(* CoDeSys 2.3.9.59 project: PD3.pro *)
(* Libraries: Standard.lib, SYSLIBCALLBACK.LIB *)

(* PLC configuration (modules and I/O channels)
Configuration EC4P-200 [Root] node -1, in %IB0 out %QB0 {EC4P_RestartPwrOn = WARMSTART; EC4P_MaxCycleTime = 20; EC4P_Com1BaudRate = 38400; EC4P_CAN1BaudRate = 125KBaud; EC4P_RoutingId = 127; EC4P_EasyNetId = 1; EC4P_EasyNetCfg = 0; EC4P_EasyNetCycleTime = 50; EC4P_RoutingChannel = CAN1; EC4P_IPFlags = 0; EC4P_IPAddress = 0; EC4P_SubNetMask = 0; EC4P_DefaultGateway = 0; EC4P_SummerWinterFlags = 0; EC4P_SummerWinterRule1 = 0; EC4P_SummerWinterRule2 = 0}
  Local I/O [EC4P_LocalIO] node 0, in %IB0 out %QB0 {EC4P_LocalInt = 0}
    I1 AT %IX0.0 [LocalBitInput] Input I1
    I2 AT %IX0.1 [LocalBitInput] Input I2
    I3 AT %IX0.2 [LocalBitInput] Input I3
    I4 AT %IX0.3 [LocalBitInput] Input I4
    I5 AT %IX0.4 [LocalBitInput] Input I5
    I6 AT %IX0.5 [LocalBitInput] Input I6
    I7 AT %IX0.6 [LocalBitInput] Input I7
    I8 AT %IX0.7 [LocalBitInput] Input I8
    I9 AT %IX1.0 [LocalBitInput] Input I9
    I10 AT %IX1.1 [LocalBitInput] Input I10
    I11 AT %IX1.2 [LocalBitInput] Input I11
    I12 AT %IX1.3 [LocalBitInput] Input I12
    I13 AT %IX1.4 [LocalDiagInput] Diagnostic Input I13
    I14 AT %IX1.5 [LocalDiagInput] Diagnostic Input I14
    I15 AT %IX1.6 [LocalDiagInput] Diagnostic Input I15
    I16 AT %IX1.7 [LocalDiagInput] Diagnostic Input I16
    I7_Analog AT %IW2 [LocalAnalogIn] Input I7, 10Bit, 0-10VDC
    I8_Analog AT %IW4 [LocalAnalogIn] Input I8, 10Bit, 0-10VDC
    I11_Analog AT %IW6 [LocalAnalogIn] Input I11, 10Bit, 0-10VDC
    I12_Analog AT %IW8 [LocalAnalogIn] Input I12, 10Bit, 0-10VDC
    Transistor Outputs [EC4P_TOutputs] node 0, in %IB10 out %QB0
      Q1 AT %QX0.0 [LocalBitOutput] Transistor-Output Q1
      Q2 AT %QX0.1 [LocalBitOutput] Transistor-Output Q2
      Q3 AT %QX0.2 [LocalBitOutput] Transistor-Output Q3
      Q4 AT %QX0.3 [LocalBitOutput] Transistor-Output Q4
      Q5 AT %QX0.4 [LocalBitOutput] Transistor-Output Q5
      Q6 AT %QX0.5 [LocalBitOutput] Transistor-Output Q6
      Q7 AT %QX0.6 [LocalBitOutput] Transistor-Output Q7
      Q8 AT %QX0.7 [LocalBitOutput] Transistor-Output Q8
    No Analog Output [EC4P_NoAnalogOutput] node 1, in %IB10 out %QB1
    No Keys [EC4P_NoKeys] node 2, in %IB10 out %QB1
    No Counter [EC4P_NoCounter] node 3, in %IB10 out %QB1
  Extension [EC4P_Extension] node 1, in %IB10 out %QB1
    No Extension [EC4P_NoExtension] node 0, in %IB10 out %QB1
*)

(* POU PLC_PRG, LD *)
PROGRAM PLC_PRG
VAR
	A: BOOL;
	B: BOOL;
	C: BOOL;
	D: BOOL;
	E: BOOL;
	ctu1: CTU;
	counter: INT;
	timer: BOOL;
	res: BOOL;
	TON1: TON;
	init: BOOL;
	tim: BOOL;
	TON2: TON;
	TON3: TON;
	temp: BOOL;
	t1: TIME;
	t2: TIME;
	TOF1: TOF;
	set_1: BOOL;
	set_2: BOOL;
	set_3: BOOL;
	set_4: BOOL;
	set_5: BOOL;
END_VAR
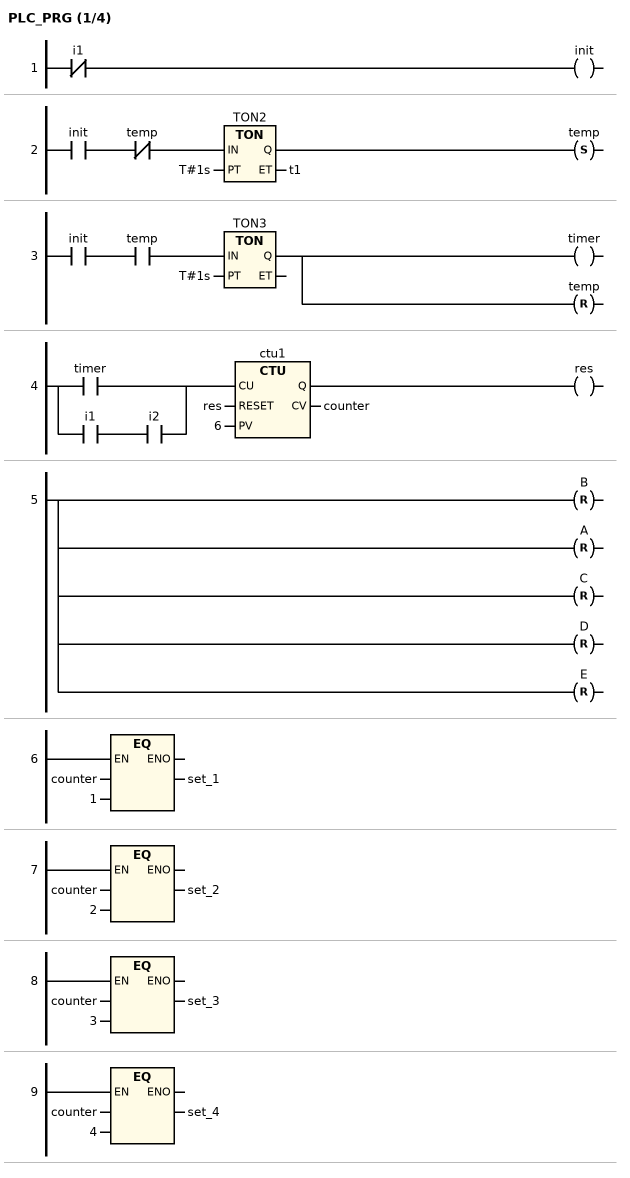
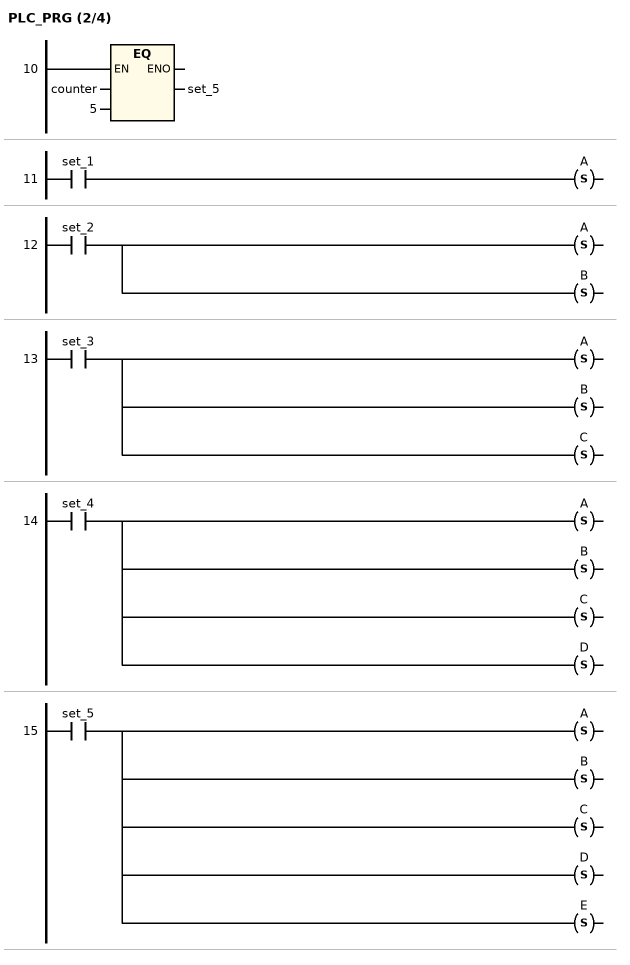
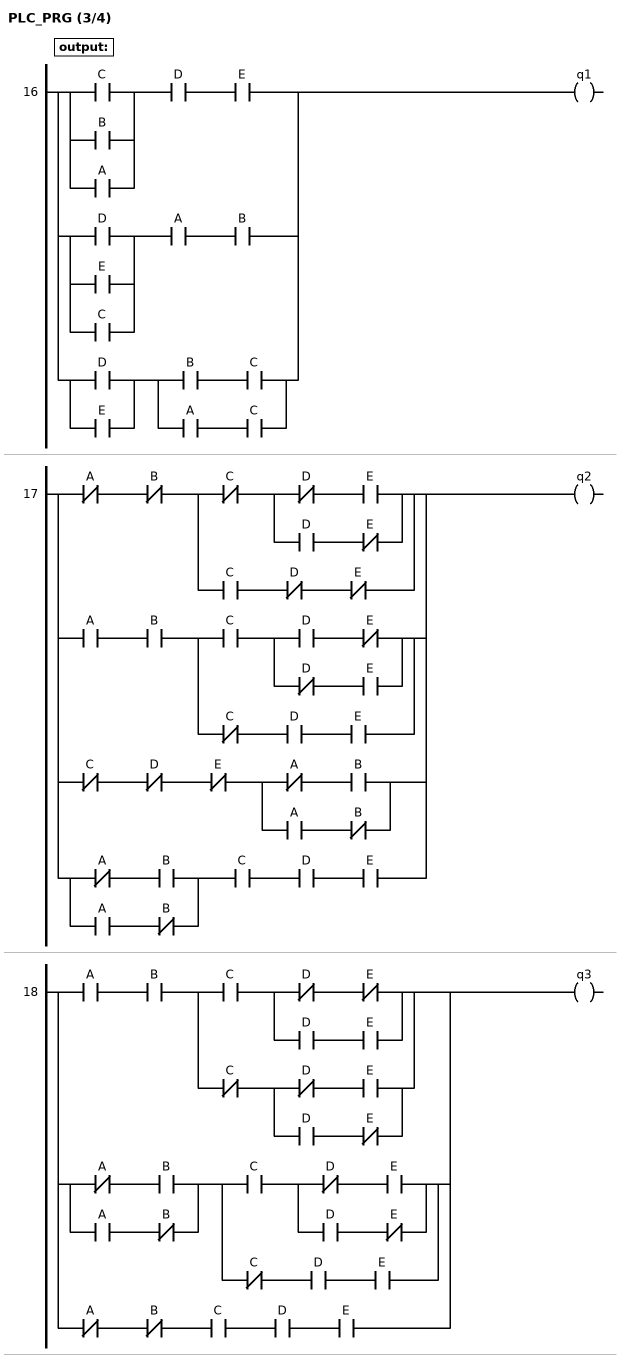
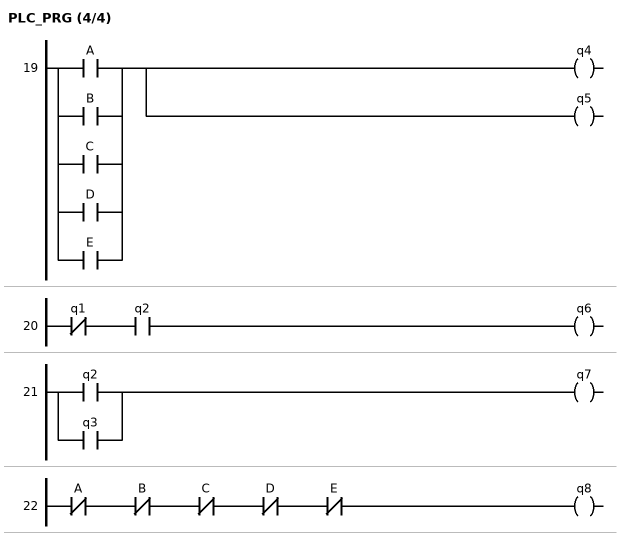
_LD_ (* Ladder Diagram *)
NETWORK 1
	[/i1] --- (init)
NETWORK 2
	[init] - [/temp] - TON2:TON(IN: *, PT: T#1s, ET => t1) --- (S temp)
NETWORK 3
	[init] - [temp] - TON3:TON(IN: *, PT: T#1s) --- (timer) (R temp)
NETWORK 4
	{ [timer] | [i1] - [i2] } - ctu1:CTU(CU: *, RESET: res, PV: 6, CV => counter) --- (res)
NETWORK 5
	* --- (R B) (R A) (R C) (R D) (R E)
NETWORK 6
	*
		EN --- EQ(counter, 1) => set_1
NETWORK 7
	*
		EN --- EQ(counter, 2) => set_2
NETWORK 8
	*
		EN --- EQ(counter, 3) => set_3
NETWORK 9
	*
		EN --- EQ(counter, 4) => set_4
NETWORK 10
	*
		EN --- EQ(counter, 5) => set_5
NETWORK 11
	[set_1] --- (S A)
NETWORK 12
	[set_2] --- (S A) (S B)
NETWORK 13
	[set_3] --- (S A) (S B) (S C)
NETWORK 14
	[set_4] --- (S A) (S B) (S C) (S D)
NETWORK 15
	[set_5] --- (S A) (S B) (S C) (S D) (S E)
NETWORK 16 output::
	{ { [C] | [B] | [A] } - [D] - [E] | { [D] | [E] | [C] } - [A] - [B] | { [D] | [E] } - { [B] - [C] | [A] - [C] } } --- (q1)
NETWORK 17
	{ [/A] - [/B] - { [/C] - { [/D] - [E] | [D] - [/E] } | [C] - [/D] - [/E] } | [A] - [B] - { [C] - { [D] - [/E] | [/D] - [E] } | [/C] - [D] - [E] } | [/C] - [/D] - [/E] - { [/A] - [B] | [A] - [/B] } | { [/A] - [B] | [A] - [/B] } - [C] - [D] - [E] } --- (q2)
NETWORK 18
	{ [A] - [B] - { [C] - { [/D] - [/E] | [D] - [E] } | [/C] - { [/D] - [E] | [D] - [/E] } } | { [/A] - [B] | [A] - [/B] } - { [C] - { [/D] - [E] | [D] - [/E] } | [/C] - [D] - [E] } | [/A] - [/B] - [C] - [D] - [E] } --- (q3)
NETWORK 19
	{ [A] | [B] | [C] | [D] | [E] } --- (q4) (q5)
NETWORK 20
	[/q1] - [q2] --- (q6)
NETWORK 21
	{ [q2] | [q3] } --- (q7)
NETWORK 22
	[/A] - [/B] - [/C] - [/D] - [/E] --- (q8)
_END_LD_
(* the same logic as Structured Text *)
(* Network 1 *)
init := NOT i1;
(* Network 2 *)
TON2(IN := init AND NOT temp, PT := T#1s);
t1 := TON2.ET;
IF TON2.Q THEN temp := TRUE; END_IF;
(* Network 3 *)
TON3(IN := init AND temp, PT := T#1s);
timer := TON3.Q;
IF TON3.Q THEN temp := FALSE; END_IF;
(* Network 4 *)
ctu1(CU := timer OR i1 AND i2, RESET := res, PV := 6);
counter := ctu1.CV;
res := ctu1.Q;
(* Network 5 *)
B := FALSE;
A := FALSE;
C := FALSE;
D := FALSE;
E := FALSE;
(* Network 6 *)
set_1 := counter = 1;
(* Network 7 *)
set_2 := counter = 2;
(* Network 8 *)
set_3 := counter = 3;
(* Network 9 *)
set_4 := counter = 4;
(* Network 10 *)
set_5 := counter = 5;
(* Network 11 *)
IF set_1 THEN A := TRUE; END_IF;
(* Network 12 *)
IF set_2 THEN A := TRUE; B := TRUE; END_IF;
(* Network 13 *)
IF set_3 THEN A := TRUE; B := TRUE; C := TRUE; END_IF;
(* Network 14 *)
IF set_4 THEN A := TRUE; B := TRUE; C := TRUE; D := TRUE; END_IF;
(* Network 15 *)
IF set_5 THEN A := TRUE; B := TRUE; C := TRUE; D := TRUE; E := TRUE; END_IF;
(* Network 16 *)
(* label: output: *)
q1 := (C OR B OR A) AND D AND E OR (D OR E OR C) AND A AND B OR (D OR E) AND (B AND C OR A AND C);
(* Network 17 *)
q2 := NOT A AND NOT B AND (NOT C AND (NOT D AND E OR D AND NOT E) OR C AND NOT D AND NOT E) OR A AND B AND (C AND (D AND NOT E OR NOT D AND E) OR NOT C AND D AND E) OR NOT C AND NOT D AND NOT E AND (NOT A AND B OR A AND NOT B) OR (NOT A AND B OR A AND NOT B) AND C AND D AND E;
(* Network 18 *)
q3 := A AND B AND (C AND (NOT D AND NOT E OR D AND E) OR NOT C AND (NOT D AND E OR D AND NOT E)) OR (NOT A AND B OR A AND NOT B) AND (C AND (NOT D AND E OR D AND NOT E) OR NOT C AND D AND E) OR NOT A AND NOT B AND C AND D AND E;
(* Network 19 *)
q4 := A OR B OR C OR D OR E;
q5 := q4;
(* Network 20 *)
q6 := NOT q1 AND q2;
(* Network 21 *)
q7 := q2 OR q3;
(* Network 22 *)
q8 := NOT A AND NOT B AND NOT C AND NOT D AND NOT E;
END_PROGRAM

(* Visualisation seg_7
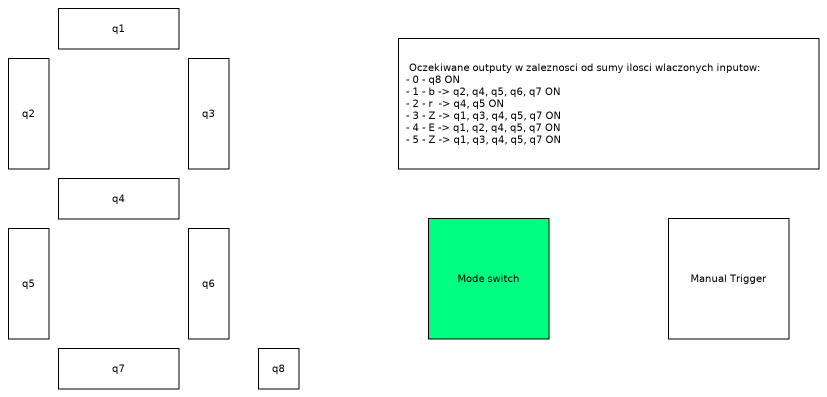
rectangle at (130,30)-(251,71): text "q1"; alarm colour if q1; toggles q1
rectangle at (260,80)-(301,191): text "q3"; alarm colour if q3; toggles q3
rectangle at (80,80)-(121,191): text "q2"; alarm colour if q2; toggles q2
rectangle at (130,200)-(251,241): text "q4"; alarm colour if q4; toggles q4
rectangle at (260,250)-(301,361): text "q6"; alarm colour if q6; toggles q6
rectangle at (80,250)-(121,361): text "q5"; alarm colour if q5; toggles q5
rectangle at (130,370)-(251,411): text "q7"; alarm colour if q7; toggles q7
rectangle at (330,370)-(371,411): text "q8"; alarm colour if q8; toggles q8
rectangle at (500,240)-(621,361): text "Mode switch"; alarm colour if i1; toggles i1
rectangle at (740,240)-(861,361): text "Manual Trigger"; alarm colour if i2; taps i2
rectangle at (470,60)-(891,191): text "Oczekiwane outputy w zaleznosci od sumy ilosci wlaczonych inputow: / - 0 - q8 ON / - 1 - b -> q2, q4, q5, q6, q7 ON / - 2 - r  -> q4, q5 ON / - 3 - Z -> q1, q3, q4, q5, q7 ON / - 4 - E -> q1, q2, q4, q5, q7 ON / - 5 - Z -> q1, q3, q4, q5, q7 ON"
*)
